TYPE ST180_PnpHorPos_e : ST110_PnpHorPos_e;
END_TYPE

(* stored: Version 1.1.0.1, ProductVersion 3.1.4024.6
   DUT ST180_PnpHorPos_e: Id {599eed5c-acee-45d6-8331-565ce1e7e09a} *)
